Omron CX-Programmer project NewProject (CX-Programmer 9.72)

# PLC NodeA: CP2E-N N

## Global symbols (name address type ; comment)
D9000 CHANNEL  ; NodeB_ErrorCode
D9001 CHANNEL  ; NodeC_Errorcode
D9002 CHANNEL  ; NodeD_ErrorCode
W10.00 BOOL  ; NodeB_link
W10.01 BOOL  ; NodeB_BUSY
W10.02 BOOL  ; NodeB_OK
W10.03 BOOL  ; NodeB_NG
W11.00 BOOL  ; NodeC_link
W11.01 BOOL  ; NodeC_BUSY
W11.02 BOOL  ; NodeC_OK
W11.03 BOOL  ; NodeC_NG
W12.00 BOOL  ; NodeD_link
W12.01 BOOL  ; NodeD_BUSY
W12.02 BOOL  ; NodeD_OK
W12.03 BOOL  ; NodeD_NG
Send_NodeB _CPxx001_SendData
Send_NodeC _CPxx001_SendData
Send_NodeD _CPxx001_SendData

## Program NewProgram1 (cyclic task 0)

### Section Section1

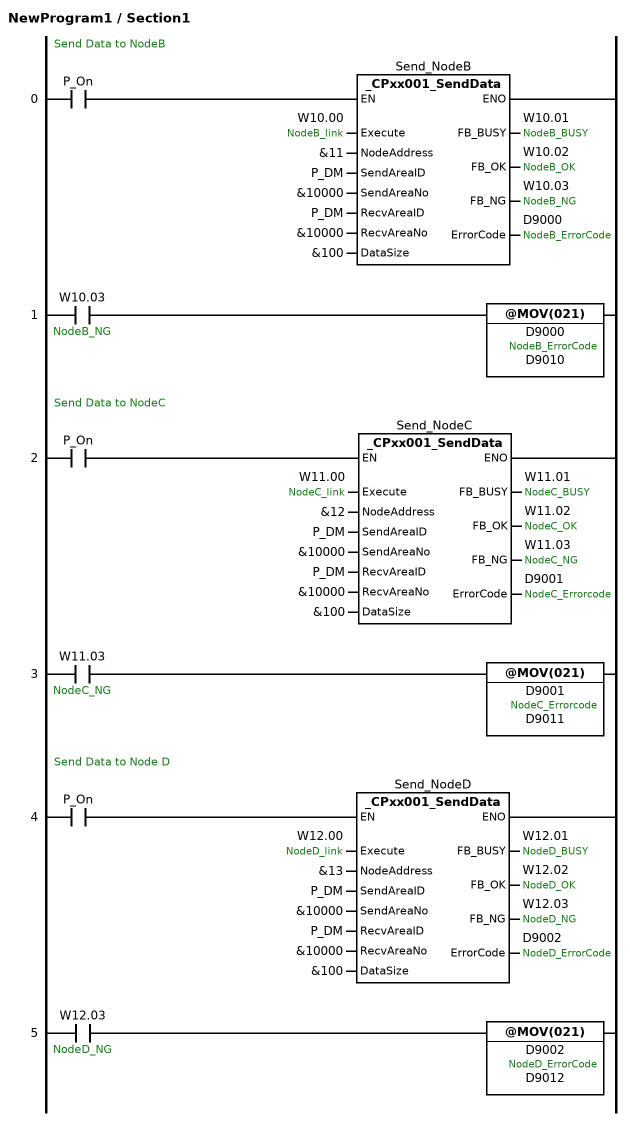
; rung 0: Send Data to NodeB
LD P_On
CALL Send_NodeB : _CPxx001_SendData (Execute := W10.00, NodeAddress := &11, SendAreaID := P_DM, SendAreaNo := &10000, RecvAreaID := P_DM, RecvAreaNo := &10000, DataSize := &100, FB_BUSY => W10.01, FB_OK => W10.02, FB_NG => W10.03, ErrorCode => D9000)  ; NodeB_link, NodeB_BUSY, NodeB_OK, NodeB_NG, NodeB_ErrorCode
; rung 1
LD W10.03  ; NodeB_NG
@MOV(021) D9000 D9010  ; NodeB_ErrorCode
; rung 2: Send Data to NodeC
LD P_On
CALL Send_NodeC : _CPxx001_SendData (Execute := W11.00, NodeAddress := &12, SendAreaID := P_DM, SendAreaNo := &10000, RecvAreaID := P_DM, RecvAreaNo := &10000, DataSize := &100, FB_BUSY => W11.01, FB_OK => W11.02, FB_NG => W11.03, ErrorCode => D9001)  ; NodeC_link, NodeC_BUSY, NodeC_OK, NodeC_NG, NodeC_Errorcode
; rung 3
LD W11.03  ; NodeC_NG
@MOV(021) D9001 D9011  ; NodeC_Errorcode
; rung 4: Send Data to Node D
LD P_On
CALL Send_NodeD : _CPxx001_SendData (Execute := W12.00, NodeAddress := &13, SendAreaID := P_DM, SendAreaNo := &10000, RecvAreaID := P_DM, RecvAreaNo := &10000, DataSize := &100, FB_BUSY => W12.01, FB_OK => W12.02, FB_NG => W12.03, ErrorCode => D9002)  ; NodeD_link, NodeD_BUSY, NodeD_OK, NodeD_NG, NodeD_ErrorCode
; rung 5
LD W12.03  ; NodeD_NG
@MOV(021) D9002 D9012  ; NodeD_ErrorCode

### Section END
; rung 0
END(001)

## Function block _CPxx001_SendData (Omron library block, body left out)

# PLC NodeB: CP2E-N N

## Global symbols (name address type ; comment)
D9000 CHANNEL  ; NodeA_ErrorCode
D9001 CHANNEL  ; NodeC_Errorcode
D9002 CHANNEL  ; NodeD_ErrorCode
W10.00 BOOL  ; NodeA_link
W10.01 BOOL  ; NodeA_BUSY
W10.02 BOOL  ; NodeA_OK
W10.03 BOOL  ; NodeA_NG
W11.00 BOOL  ; NodeC_link
W11.01 BOOL  ; NodeC_BUSY
W11.02 BOOL  ; NodeC_OK
W11.03 BOOL  ; NodeC_NG
W12.00 BOOL  ; NodeD_link
W12.01 BOOL  ; NodeD_BUSY
W12.02 BOOL  ; NodeD_OK
W12.03 BOOL  ; NodeD_NG
Send_NodeA _CPxx001_SendData
Send_NodeC _CPxx001_SendData
Send_NodeD _CPxx001_SendData

## Program NewProgram1 (cyclic task 0)

### Section Section1

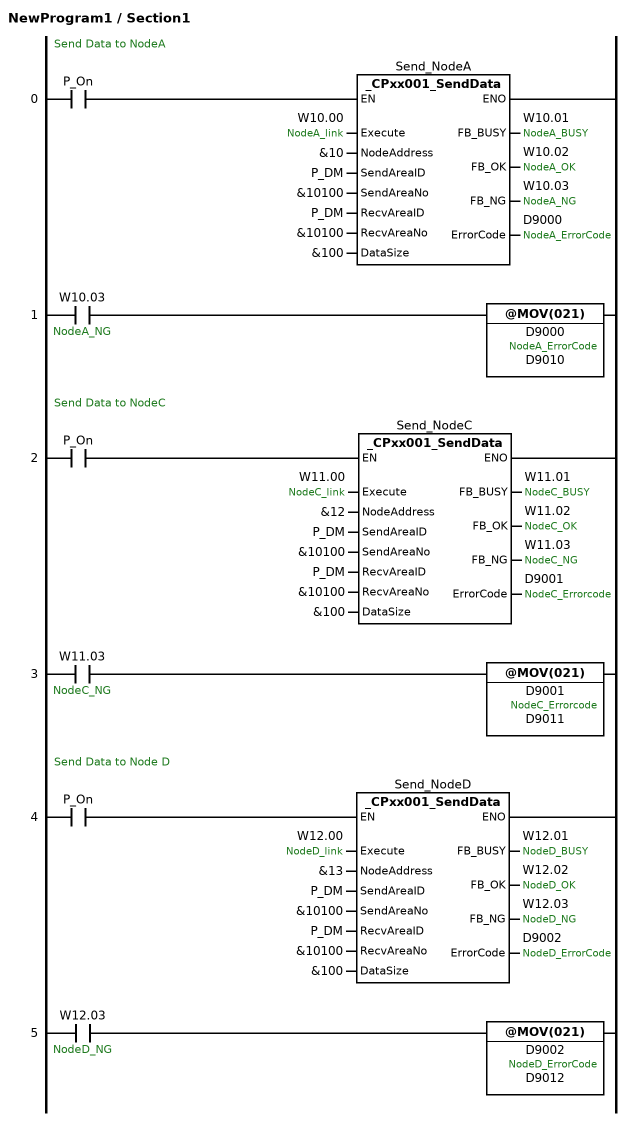
; rung 0: Send Data to NodeA
LD P_On
CALL Send_NodeA : _CPxx001_SendData (Execute := W10.00, NodeAddress := &10, SendAreaID := P_DM, SendAreaNo := &10100, RecvAreaID := P_DM, RecvAreaNo := &10100, DataSize := &100, FB_BUSY => W10.01, FB_OK => W10.02, FB_NG => W10.03, ErrorCode => D9000)  ; NodeA_link, NodeA_BUSY, NodeA_OK, NodeA_NG, NodeA_ErrorCode
; rung 1
LD W10.03  ; NodeA_NG
@MOV(021) D9000 D9010  ; NodeA_ErrorCode
; rung 2: Send Data to NodeC
LD P_On
CALL Send_NodeC : _CPxx001_SendData (Execute := W11.00, NodeAddress := &12, SendAreaID := P_DM, SendAreaNo := &10100, RecvAreaID := P_DM, RecvAreaNo := &10100, DataSize := &100, FB_BUSY => W11.01, FB_OK => W11.02, FB_NG => W11.03, ErrorCode => D9001)  ; NodeC_link, NodeC_BUSY, NodeC_OK, NodeC_NG, NodeC_Errorcode
; rung 3
LD W11.03  ; NodeC_NG
@MOV(021) D9001 D9011  ; NodeC_Errorcode
; rung 4: Send Data to Node D
LD P_On
CALL Send_NodeD : _CPxx001_SendData (Execute := W12.00, NodeAddress := &13, SendAreaID := P_DM, SendAreaNo := &10100, RecvAreaID := P_DM, RecvAreaNo := &10100, DataSize := &100, FB_BUSY => W12.01, FB_OK => W12.02, FB_NG => W12.03, ErrorCode => D9002)  ; NodeD_link, NodeD_BUSY, NodeD_OK, NodeD_NG, NodeD_ErrorCode
; rung 5
LD W12.03  ; NodeD_NG
@MOV(021) D9002 D9012  ; NodeD_ErrorCode

### Section END
; rung 0
END(001)

## Function block _CPxx001_SendData (Omron library block, body left out)

# PLC NodeC: CP2E-N N

## Global symbols (name address type ; comment)
D9000 CHANNEL  ; NodeA_ErrorCode
D9001 CHANNEL  ; NodeB_Errorcode
D9002 CHANNEL  ; NodeD_ErrorCode
W10.00 BOOL  ; NodeA_link
W10.01 BOOL  ; NodeA_BUSY
W10.02 BOOL  ; NodeA_OK
W10.03 BOOL  ; NodeA_NG
W11.00 BOOL  ; NodeB_link
W11.01 BOOL  ; NodeB_BUSY
W11.02 BOOL  ; NodeB_OK
W11.03 BOOL  ; NodeB_NG
W12.00 BOOL  ; NodeD_link
W12.01 BOOL  ; NodeD_BUSY
W12.02 BOOL  ; NodeD_OK
W12.03 BOOL  ; NodeD_NG
Send_NodeA _CPxx001_SendData
Send_NodeB _CPxx001_SendData
Send_NodeD _CPxx001_SendData

## Program NewProgram1 (cyclic task 0)

### Section Section1

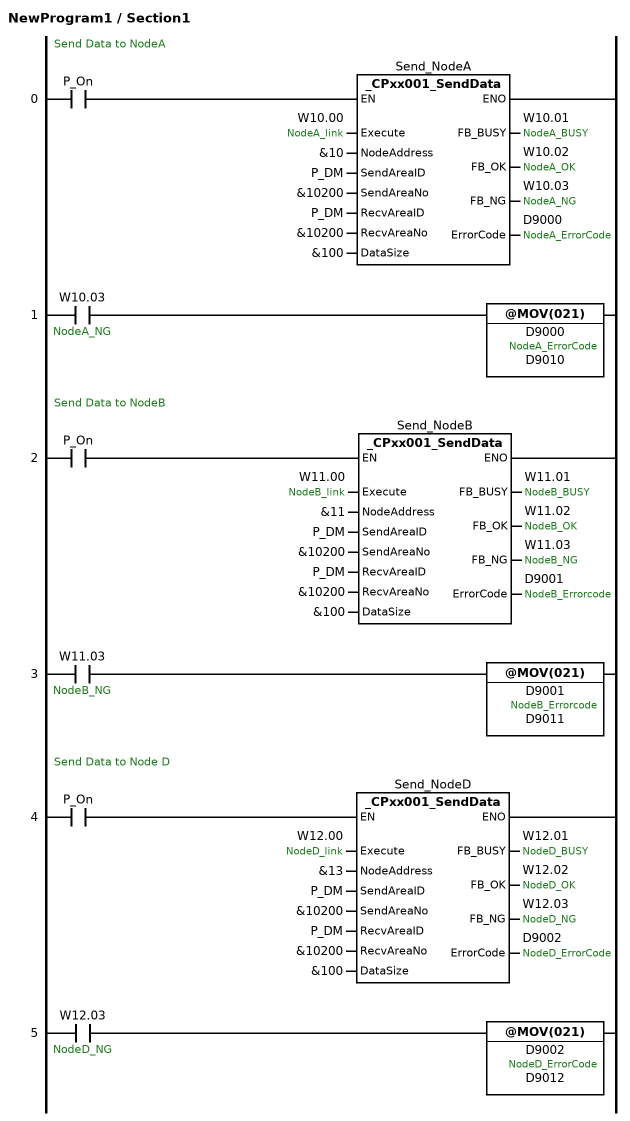
; rung 0: Send Data to NodeA
LD P_On
CALL Send_NodeA : _CPxx001_SendData (Execute := W10.00, NodeAddress := &10, SendAreaID := P_DM, SendAreaNo := &10200, RecvAreaID := P_DM, RecvAreaNo := &10200, DataSize := &100, FB_BUSY => W10.01, FB_OK => W10.02, FB_NG => W10.03, ErrorCode => D9000)  ; NodeA_link, NodeA_BUSY, NodeA_OK, NodeA_NG, NodeA_ErrorCode
; rung 1
LD W10.03  ; NodeA_NG
@MOV(021) D9000 D9010  ; NodeA_ErrorCode
; rung 2: Send Data to NodeB
LD P_On
CALL Send_NodeB : _CPxx001_SendData (Execute := W11.00, NodeAddress := &11, SendAreaID := P_DM, SendAreaNo := &10200, RecvAreaID := P_DM, RecvAreaNo := &10200, DataSize := &100, FB_BUSY => W11.01, FB_OK => W11.02, FB_NG => W11.03, ErrorCode => D9001)  ; NodeB_link, NodeB_BUSY, NodeB_OK, NodeB_NG, NodeB_Errorcode
; rung 3
LD W11.03  ; NodeB_NG
@MOV(021) D9001 D9011  ; NodeB_Errorcode
; rung 4: Send Data to Node D
LD P_On
CALL Send_NodeD : _CPxx001_SendData (Execute := W12.00, NodeAddress := &13, SendAreaID := P_DM, SendAreaNo := &10200, RecvAreaID := P_DM, RecvAreaNo := &10200, DataSize := &100, FB_BUSY => W12.01, FB_OK => W12.02, FB_NG => W12.03, ErrorCode => D9002)  ; NodeD_link, NodeD_BUSY, NodeD_OK, NodeD_NG, NodeD_ErrorCode
; rung 5
LD W12.03  ; NodeD_NG
@MOV(021) D9002 D9012  ; NodeD_ErrorCode

### Section END
; rung 0
END(001)

## Function block _CPxx001_SendData (Omron library block, body left out)

# PLC NodeD: CP2E-N N

## Global symbols (name address type ; comment)
D9000 CHANNEL  ; NodeA_ErrorCode
D9001 CHANNEL  ; NodeB_Errorcode
D9002 CHANNEL  ; NodeC_ErrorCode
W10.00 BOOL  ; NodeA_link
W10.01 BOOL  ; NodeA_BUSY
W10.02 BOOL  ; NodeA_OK
W10.03 BOOL  ; NodeA_NG
W11.00 BOOL  ; NodeB_link
W11.01 BOOL  ; NodeB_BUSY
W11.02 BOOL  ; NodeB_OK
W11.03 BOOL  ; NodeB_NG
W12.00 BOOL  ; NodeC_link
W12.01 BOOL  ; NodeC_BUSY
W12.02 BOOL  ; NodeC_OK
W12.03 BOOL  ; NodeC_NG
Send_NodeA _CPxx001_SendData
Send_NodeB _CPxx001_SendData
Send_NodeC _CPxx001_SendData

## Program NewProgram1 (cyclic task 0)

### Section Section1

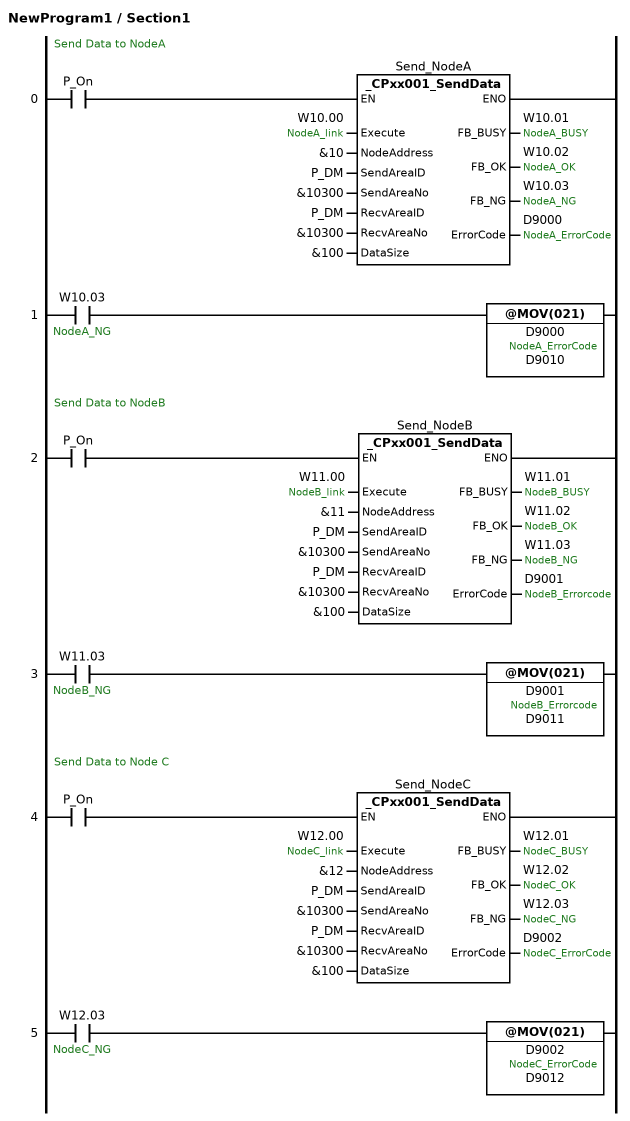
; rung 0: Send Data to NodeA
LD P_On
CALL Send_NodeA : _CPxx001_SendData (Execute := W10.00, NodeAddress := &10, SendAreaID := P_DM, SendAreaNo := &10300, RecvAreaID := P_DM, RecvAreaNo := &10300, DataSize := &100, FB_BUSY => W10.01, FB_OK => W10.02, FB_NG => W10.03, ErrorCode => D9000)  ; NodeA_link, NodeA_BUSY, NodeA_OK, NodeA_NG, NodeA_ErrorCode
; rung 1
LD W10.03  ; NodeA_NG
@MOV(021) D9000 D9010  ; NodeA_ErrorCode
; rung 2: Send Data to NodeB
LD P_On
CALL Send_NodeB : _CPxx001_SendData (Execute := W11.00, NodeAddress := &11, SendAreaID := P_DM, SendAreaNo := &10300, RecvAreaID := P_DM, RecvAreaNo := &10300, DataSize := &100, FB_BUSY => W11.01, FB_OK => W11.02, FB_NG => W11.03, ErrorCode => D9001)  ; NodeB_link, NodeB_BUSY, NodeB_OK, NodeB_NG, NodeB_Errorcode
; rung 3
LD W11.03  ; NodeB_NG
@MOV(021) D9001 D9011  ; NodeB_Errorcode
; rung 4: Send Data to Node C
LD P_On
CALL Send_NodeC : _CPxx001_SendData (Execute := W12.00, NodeAddress := &12, SendAreaID := P_DM, SendAreaNo := &10300, RecvAreaID := P_DM, RecvAreaNo := &10300, DataSize := &100, FB_BUSY => W12.01, FB_OK => W12.02, FB_NG => W12.03, ErrorCode => D9002)  ; NodeC_link, NodeC_BUSY, NodeC_OK, NodeC_NG, NodeC_ErrorCode
; rung 5
LD W12.03  ; NodeC_NG
@MOV(021) D9002 D9012  ; NodeC_ErrorCode

### Section END
; rung 0
END(001)

## Function block _CPxx001_SendData (Omron library block, body left out)